{attribute 'qualified_only'}
VAR_GLOBAL
	bWinchEnable	: BOOL;
	bCylEnable 		: BOOL;
	stAutomaticControlSettingsWinch 			: ST_AutomaticControlSettings;
	stMotionReferenceGeneratorSettingsWinch  	: ST_MotionReferenceGeneratorSettings;
	stAutomaticControlSettingsCylinder 			: ST_AutomaticControlSettings;
	stMotionReferenceGeneratorSettingsCylinder  : ST_MotionReferenceGeneratorSettings;
	stModifyAutomaticControlSettingsWinch 		: ST_ModifyAutomaticControlSettings;
	stModifyAutomaticControlSettingsCylinder 	: ST_ModifyAutomaticControlSettings;
END_VAR

(* stored: Version 1.1.0.1, ProductVersion 3.1.4024.11
   GVL G_Hmi: Id {2bbce215-5f34-4630-bf6a-024acf95f838} *)
